(* PLC project  *)

PROGRAM P

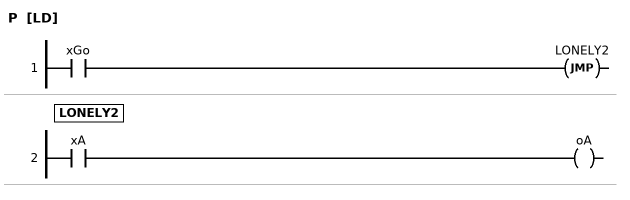
(* LD diagram, written out as Structured Text *)
IF xGo THEN JMP LONELY2; END_IF;
LONELY1:
LONELY2:
oA := xA;
END_PROGRAM
